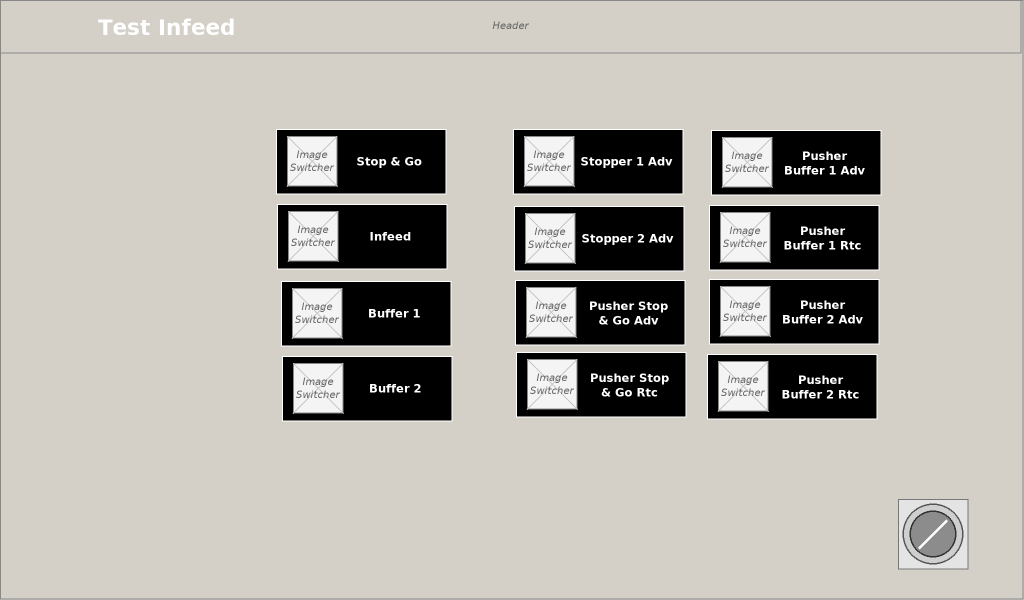
VISUALIZATION Test_Infeed  // 1024x600
    Frame (0,-2 1021x55)
        shows Header()
    Label (95,15 250x25), "Test Infeed"
    RotarySwitch (898,499 70x70), variable: HMI_GVL.bTestModeEnableInfeed, behaviour: TOGGLE, style: Switch-RotarySwitch-Gray
    RoundedRectangle (276,129 170x65)
        toggle HMI_GVL.Test_BoxStopGo_Fwd
    Label (321,149 137x25), "Stop & Go"
    ImageSwitcher (287,136 50x50), variable: HMI_GVL.Test_BoxStopGo_Fwd, behaviour: TOGGLE
    RoundedRectangle (513,129 170x65)
        toggle HMI_GVL.Test_Stopper1
    Label (558,149 137x25), "Stopper 1 Adv"
    ImageSwitcher (524,136 50x50), variable: HMI_GVL.Test_Stopper1, behaviour: TOGGLE
    RoundedRectangle (514,206 170x65)
        toggle HMI_GVL.Test_Stopper2
    Label (559,226 137x25), "Stopper 2 Adv"
    ImageSwitcher (525,213 50x50), variable: HMI_GVL.Test_Stopper2, behaviour: TOGGLE
    RoundedRectangle (277,204 170x65)
        toggle HMI_GVL.Test_BoxInfeed_Fwd
    Label (322,224 137x25), "Infeed"
    ImageSwitcher (288,211 50x50), variable: HMI_GVL.Test_BoxInfeed_Fwd, behaviour: TOGGLE
    RoundedRectangle (281,281 170x65)
        toggle HMI_GVL.Test_BoxBuffer1_Fwd
    Label (326,301 137x25), "Buffer 1"
    ImageSwitcher (292,288 50x50), variable: HMI_GVL.Test_BoxBuffer1_Fwd, behaviour: TOGGLE
    RoundedRectangle (282,356 170x65)
        toggle HMI_GVL.Test_BoxBuffer2_Fwd
    Label (327,376 137x25), "Buffer 2"
    ImageSwitcher (293,363 50x50), variable: HMI_GVL.Test_BoxBuffer2_Fwd, behaviour: TOGGLE
    RoundedRectangle (515,280 170x65)
        toggle HMI_GVL.Test_Pusher_StopGo_Adv
    Label (560,292 137x43), "Pusher Stop & Go Adv"
    ImageSwitcher (526,287 50x50), variable: HMI_GVL.Test_Pusher_StopGo_Adv, behaviour: TOGGLE
    RoundedRectangle (516,352 170x65)
        toggle HMI_GVL.Test_Pusher_StopGo_Rtc
    Label (561,364 137x43), "Pusher Stop & Go Rtc"
    ImageSwitcher (527,359 50x50), variable: HMI_GVL.Test_Pusher_StopGo_Rtc, behaviour: TOGGLE
    RoundedRectangle (711,130 170x65)
        toggle HMI_GVL.Test_Pusher_Buffer1_Adv
    Label (756,142 137x43), "Pusher Buffer 1 Adv"
    ImageSwitcher (722,137 50x50), variable: HMI_GVL.Test_Pusher_Buffer1_Adv, behaviour: TOGGLE
    RoundedRectangle (709,205 170x65)
        toggle HMI_GVL.Test_Pusher_Buffer1_Rtc
    Label (754,217 137x43), "Pusher Buffer 1 Rtc"
    ImageSwitcher (720,212 50x50), variable: HMI_GVL.Test_Pusher_Buffer1_Rtc, behaviour: TOGGLE
    RoundedRectangle (709,279 170x65)
        toggle HMI_GVL.Test_Pusher_Buffer2_Adv
    Label (754,291 137x43), "Pusher Buffer 2 Adv"
    ImageSwitcher (720,286 50x50), variable: HMI_GVL.Test_Pusher_Buffer2_Adv, behaviour: TOGGLE
    RoundedRectangle (707,354 170x65)
        toggle HMI_GVL.Test_Pusher_Buffer2_Rtc
    Label (752,366 137x43), "Pusher Buffer 2 Rtc"
    ImageSwitcher (718,361 50x50), variable: HMI_GVL.Test_Pusher_Buffer2_Rtc, behaviour: TOGGLE
END_VISUALIZATION

(* stored: Version 1.1.0.1, ProductVersion 3.1.4024.12
   Visu Test_Infeed: Id {3db68de9-dc34-4093-a526-fc00d445b139} *)
